Fanuc KAREL source: kb00089.KL

-- PROVISIONAL review KL for V940-1; original PC SHA256 f94441e1c34a23ecc10af7677e7ede9ef07a75c796108e25cc197d56cf80dc2a
-- Incomplete behavior may be omitted. Consult companion uncertainty JSON. Do not deploy.
PROGRAM KB00089
%NOLOCKGROUP
BEGIN
  -- V9_ZERO_TABLE_METADATA_HINT layout=0002_ascii; no indexed target words; source/name/runtime held
  -- UNRESOLVED_PC offsets 5-12; opcodes 9D,23
  -- UNRESOLVED_PC offsets 17-24; opcodes 9D,23
  -- UNRESOLVED_PC offsets 29-36; opcodes 9D,23
  -- UNRESOLVED_PC offsets 41-48; opcodes 9D,23
  -- UNRESOLVED_PC offsets 53-60; opcodes 9D,23
  -- UNRESOLVED_PC offsets 65-72; opcodes 9D,23
  -- UNRESOLVED_PC offsets 77-117; opcodes 27,22,22,22,22,22,22,31
  -- UNRESOLVED_PC offsets 122-126; opcodes 7F
END KB00089
